// TIA Portal V16 program export: 1 tag tables, 0 data types, 1 data blocks, 11 code blocks (in call order from the OBs), 6 instance data blocks

VAR_GLOBAL   // PLC tag table "Standard-Variablentabelle"
   "Belt Conveyor (4m) 0 Encoder Signal A" AT %I0.0 : Bool;
   "Retroreflective Sensor 0" AT %I0.1 : Bool;
   "Retroreflective Sensor 1" AT %I0.2 : Bool;
   "Diffuse Sensor 0" AT %I0.3 : Bool;
   Clock_Byte AT %MB0 : Byte;
   Clock_10Hz AT %M0.0 : Bool;
   Clock_5Hz AT %M0.1 : Bool;
   "Clock_2.5Hz" AT %M0.2 : Bool;
   Clock_2Hz AT %M0.3 : Bool;
   "Clock_1.25Hz" AT %M0.4 : Bool;
   Clock_1Hz AT %M0.5 : Bool;
   "Clock_0.625Hz" AT %M0.6 : Bool;
   "Clock_0.5Hz" AT %M0.7 : Bool;
   "Diffuse Sensor 1" AT %I0.4 : Bool;
   "Diffuse Sensor 2" AT %I0.5 : Bool;
   "Diffuse Sensor 3" AT %I0.6 : Bool;
   "Belt Conveyor (2m) 0" AT %Q0.0 : Bool;
   "Belt Conveyor (2m) 1" AT %Q0.1 : Bool;
   "Belt Conveyor (2m) 2" AT %Q0.2 : Bool;
   "Belt Conveyor (2m) 3" AT %Q0.3 : Bool;
   "Belt Conveyor (4m) 0" AT %Q0.4 : Bool;
   "Conveyor Scale 0 (+)" AT %Q0.5 : Bool;
   "Pop Up Wheel Sorter 0 (+)" AT %Q0.6 : Bool;
   "Pop Up Wheel Sorter 0 (Left)" AT %Q0.7 : Bool;
   "Pop Up Wheel Sorter 0 (Right)" AT %Q1.0 : Bool;
   "Vision Sensor 0" AT %ID30 : DInt;
   Factory_Running AT %I0.7 : Bool;
   "Emergency Stop 0" AT %I1.0 : Bool;
   "Selector 0 (State 0)" AT %I1.1 : Bool;
   "Start Button 0" AT %I1.2 : Bool;
   "Two-Axis Pick & Place 0 (Detected)" AT %I1.3 : Bool;
   "Two-Axis Pick & Place 0 (Moving X)" AT %I1.4 : Bool;
   "Two-Axis Pick & Place 0 (Moving Z)" AT %I1.5 : Bool;
   "Two-Axis Pick & Place 0 X" AT %Q1.1 : Bool;
   "Two-Axis Pick & Place 0 Z" AT %Q1.2 : Bool;
   "Two-Axis Pick & Place 0 (Grab)" AT %Q1.3 : Bool;
   "Conveyor Scale 0 Weight (V)" AT %ID42 : Real;
   "Diffuse Sensor 4" AT %I1.6 : Bool;
   "Diffuse Sensor 6" AT %I1.7 : Bool;
   "Diffuse Sensor 5" AT %I2.0 : Bool;
   System_Byte AT %MB1 : Byte;
   FirstScan AT %M1.0 : Bool;
   DiagStatusUpdate AT %M1.1 : Bool;
   AlwaysTRUE AT %M1.2 : Bool;
   AlwaysFALSE AT %M1.3 : Bool;
END_VAR

DATA_BLOCK "DB_IO"   // DB1
{ S7_Optimized_Access := 'TRUE' }
VERSION : 0.1
// stored: AutoNumber true, IsOnlyStoredInLoadMemory false, IsRetainMemResEnabled false, IsWriteProtectedInAS false, MemoryReserve 100
   VAR
      One_shot : Array[0..10] of Bool;
      Green_position : DWord;
      Box_position : DWord;
      Green_raw_detected : Bool;
      System_running : Bool;
      StepA : Array[0..10] of Bool;
      Production_line_Init : Bool;
      System_Ready : Bool;
      Weight : Int;
      RunPickAndPlace : Bool;
      StepB : Array[0..10] of Bool;
      StepC : Array[0..10] of Bool;
      "counter" : Int;
   END_VAR
BEGIN
END_DATA_BLOCK

ORGANIZATION_BLOCK "Main"   // OB1, FBD, ProgramCycle
TITLE = "Main Program Sweep (Cycle)"
{ S7_Optimized_Access := 'TRUE' }
VERSION : 0.1
// stored: AutoNumber true, IsIECCheckEnabled false, SetENOAutomatically false
   VAR_INPUT
      Initial_Call : Bool;   // Initial call of this OB
      Remanence : Bool;   // =True, if remanent data are available
   END_VAR
BEGIN

REGION Network 1
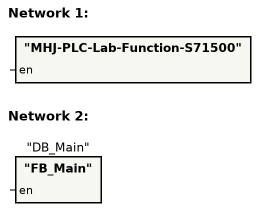
   "MHJ-PLC-Lab-Function-S71500"();
END_REGION

REGION Network 2
   "DB_Main"();   // "FB_Main"
END_REGION
END_ORGANIZATION_BLOCK

FUNCTION_BLOCK "FB_Main"   // FB2, LAD
{ S7_Optimized_Access := 'TRUE' }
VERSION : 0.1
// stored: AutoNumber true, IsIECCheckEnabled false, IsRetainMemResEnabled false, MemoryReserve 100, SetENOAutomatically false, UDAEnableTagReadback false
   VAR
      FB_Conveyor_Entry { S7_SetPoint := 'True'} : "FB_Conveyor";
      FB_Conveyor_Weight { S7_SetPoint := 'True'} : "FB_Conveyor";
      FB_WheelSorter_Instance { S7_SetPoint := 'True'} : "FB_WheelSorter";
      FB_Conveyor_Left { S7_SetPoint := 'True'} : "FB_Conveyor";
      FB_Conveyor_Straight { S7_SetPoint := 'True'} : "FB_Conveyor";
      FB_Conveyor_Right { S7_SetPoint := 'True'} : "FB_Conveyor";
      FB_PickAndPlace_Instance { S7_SetPoint := 'True'} : "FB_PickAndPlace";
      FB_Conveyor_4belt { S7_SetPoint := 'True'} : "FB_Conveyor";
   END_VAR
BEGIN

REGION Network 1
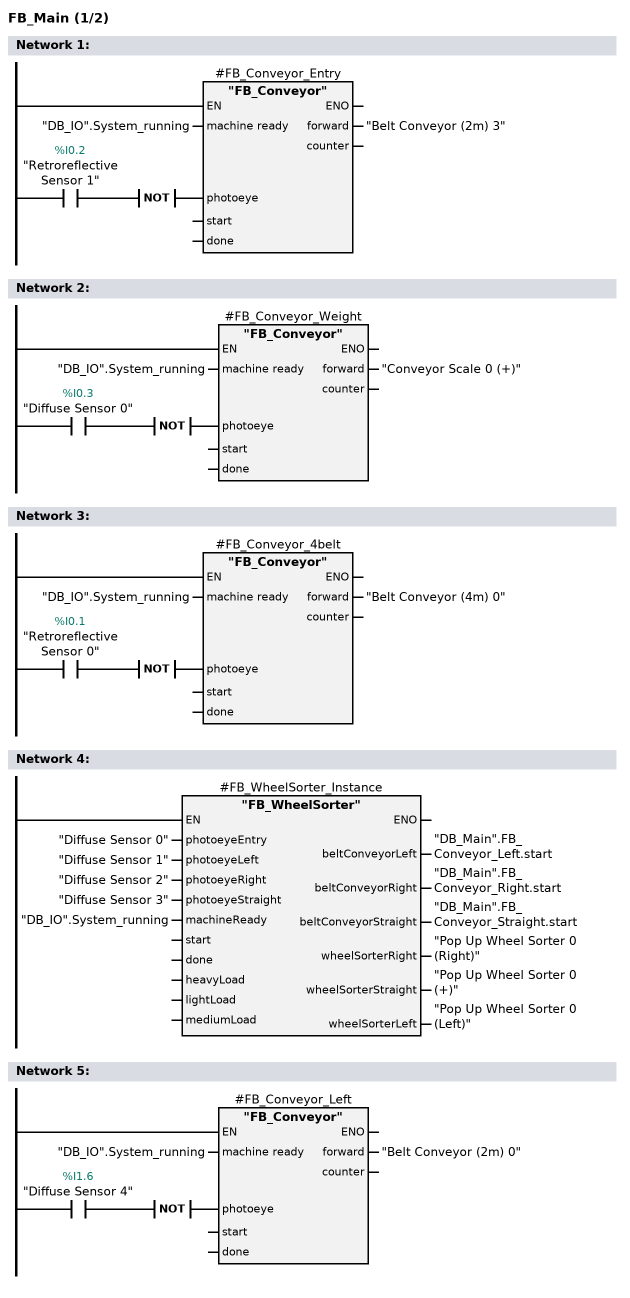
   RUNG wire#powerrail
      #FB_Conveyor_Entry(photoeye := wire#w1, "machine ready" := "DB_IO".System_running, start :=, done :=, forward => "Belt Conveyor (2m) 3", "counter" =>)
   END_RUNG
   RUNG wire#powerrail
      Contact( "Retroreflective Sensor 1" )
      Not()
   END_RUNG wire#w1
   // the same network as SCL:
   #FB_Conveyor_Entry("machine ready" := "DB_IO".System_running,   // "FB_Conveyor"
                      photoeye := NOT "Retroreflective Sensor 1",
                      forward => "Belt Conveyor (2m) 3");
END_REGION

REGION Network 2
   RUNG wire#powerrail
      #FB_Conveyor_Weight(photoeye := wire#w1, "machine ready" := "DB_IO".System_running, start :=, done :=, forward => "Conveyor Scale 0 (+)", "counter" =>)
   END_RUNG
   RUNG wire#powerrail
      Contact( "Diffuse Sensor 0" )
      Not()
   END_RUNG wire#w1
   // the same network as SCL:
   #FB_Conveyor_Weight("machine ready" := "DB_IO".System_running,   // "FB_Conveyor"
                       photoeye := NOT "Diffuse Sensor 0",
                       forward => "Conveyor Scale 0 (+)");
END_REGION

REGION Network 3
   RUNG wire#powerrail
      #FB_Conveyor_4belt(photoeye := wire#w1, "machine ready" := "DB_IO".System_running, start :=, done :=, forward => "Belt Conveyor (4m) 0", "counter" =>)
   END_RUNG
   RUNG wire#powerrail
      Contact( "Retroreflective Sensor 0" )
      Not()
   END_RUNG wire#w1
   // the same network as SCL:
   #FB_Conveyor_4belt("machine ready" := "DB_IO".System_running,   // "FB_Conveyor"
                      photoeye := NOT "Retroreflective Sensor 0",
                      forward => "Belt Conveyor (4m) 0");
END_REGION

REGION Network 4
   RUNG wire#powerrail
      #FB_WheelSorter_Instance(photoeyeEntry := "Diffuse Sensor 0", photoeyeLeft := "Diffuse Sensor 1", photoeyeRight := "Diffuse Sensor 2", photoeyeStraight := "Diffuse Sensor 3", machineReady := "DB_IO".System_running, start :=, done :=, heavyLoad :=, lightLoad :=, mediumLoad :=, beltConveyorLeft => "DB_Main".FB_Conveyor_Left.start, beltConveyorRight => "DB_Main".FB_Conveyor_Right.start, beltConveyorStraight => "DB_Main".FB_Conveyor_Straight.start, wheelSorterRight => "Pop Up Wheel Sorter 0 (Right)", wheelSorterStraight => "Pop Up Wheel Sorter 0 (+)", wheelSorterLeft => "Pop Up Wheel Sorter 0 (Left)")
   END_RUNG
   // the same network as SCL:
   #FB_WheelSorter_Instance(photoeyeEntry := "Diffuse Sensor 0",   // "FB_WheelSorter"
                           photoeyeLeft := "Diffuse Sensor 1",
                           photoeyeRight := "Diffuse Sensor 2",
                           photoeyeStraight := "Diffuse Sensor 3",
                           machineReady := "DB_IO".System_running,
                           beltConveyorLeft => "DB_Main".FB_Conveyor_Left.start,
                           beltConveyorRight => "DB_Main".FB_Conveyor_Right.start,
                           beltConveyorStraight => "DB_Main".FB_Conveyor_Straight.start,
                           wheelSorterRight => "Pop Up Wheel Sorter 0 (Right)",
                           wheelSorterStraight => "Pop Up Wheel Sorter 0 (+)",
                           wheelSorterLeft => "Pop Up Wheel Sorter 0 (Left)");
END_REGION

REGION Network 5
   RUNG wire#powerrail
      #FB_Conveyor_Left(photoeye := wire#w1, "machine ready" := "DB_IO".System_running, start :=, done :=, forward => "Belt Conveyor (2m) 0", "counter" =>)
   END_RUNG
   RUNG wire#powerrail
      Contact( "Diffuse Sensor 4" )
      Not()
   END_RUNG wire#w1
   // the same network as SCL:
   #FB_Conveyor_Left("machine ready" := "DB_IO".System_running,   // "FB_Conveyor"
                     photoeye := NOT "Diffuse Sensor 4",
                     forward => "Belt Conveyor (2m) 0");
END_REGION

REGION Network 6
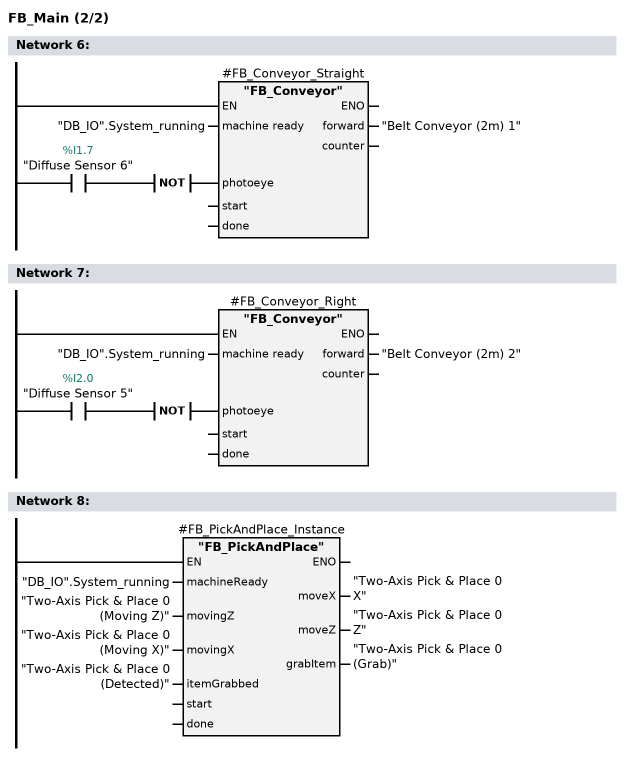
   RUNG wire#powerrail
      #FB_Conveyor_Straight(photoeye := wire#w1, "machine ready" := "DB_IO".System_running, start :=, done :=, forward => "Belt Conveyor (2m) 1", "counter" =>)
   END_RUNG
   RUNG wire#powerrail
      Contact( "Diffuse Sensor 6" )
      Not()
   END_RUNG wire#w1
   // the same network as SCL:
   #FB_Conveyor_Straight("machine ready" := "DB_IO".System_running,   // "FB_Conveyor"
                         photoeye := NOT "Diffuse Sensor 6",
                         forward => "Belt Conveyor (2m) 1");
END_REGION

REGION Network 7
   RUNG wire#powerrail
      #FB_Conveyor_Right(photoeye := wire#w1, "machine ready" := "DB_IO".System_running, start :=, done :=, forward => "Belt Conveyor (2m) 2", "counter" =>)
   END_RUNG
   RUNG wire#powerrail
      Contact( "Diffuse Sensor 5" )
      Not()
   END_RUNG wire#w1
   // the same network as SCL:
   #FB_Conveyor_Right("machine ready" := "DB_IO".System_running,   // "FB_Conveyor"
                      photoeye := NOT "Diffuse Sensor 5",
                      forward => "Belt Conveyor (2m) 2");
END_REGION

REGION Network 8
   #FB_PickAndPlace_Instance(machineReady := "DB_IO".System_running,   // "FB_PickAndPlace"
                           movingZ := "Two-Axis Pick & Place 0 (Moving Z)",
                           movingX := "Two-Axis Pick & Place 0 (Moving X)",
                           itemGrabbed := "Two-Axis Pick & Place 0 (Detected)",
                           moveX => "Two-Axis Pick & Place 0 X",
                           moveZ => "Two-Axis Pick & Place 0 Z",
                           grabItem => "Two-Axis Pick & Place 0 (Grab)");
END_REGION
END_FUNCTION_BLOCK

FUNCTION_BLOCK "FB_WheelSorter"   // FB5, LAD
{ S7_Optimized_Access := 'TRUE' }
VERSION : 0.1
// stored: AutoNumber true, IsIECCheckEnabled false, IsRetainMemResEnabled false, MemoryReserve 100, SetENOAutomatically false, UDAEnableTagReadback false
   VAR_INPUT
      photoeyeEntry : Bool;
      photoeyeLeft : Bool;
      photoeyeRight : Bool;
      photoeyeStraight : Bool;
      machineReady : Bool;
   END_VAR
   VAR_OUTPUT
      beltConveyorLeft : Bool;
      beltConveyorRight : Bool;
      beltConveyorStraight : Bool;
      wheelSorterRight : Bool;
      wheelSorterStraight : Bool;
      wheelSorterLeft : Bool;
   END_VAR
   VAR_IN_OUT
      start : Bool;
      done : Bool;
      heavyLoad : Bool := false;
      lightLoad : Bool := false;
      mediumLoad : Bool := false;
   END_VAR
   VAR
      "step" : Array[0..20] of Bool;
   END_VAR
   VAR_TEMP   // added for the SCL form of the ladder/FBD networks
      _w1 : Bool;
      _w2 : Bool;
      _w3 : Bool;
   END_VAR
BEGIN

REGION Network 1
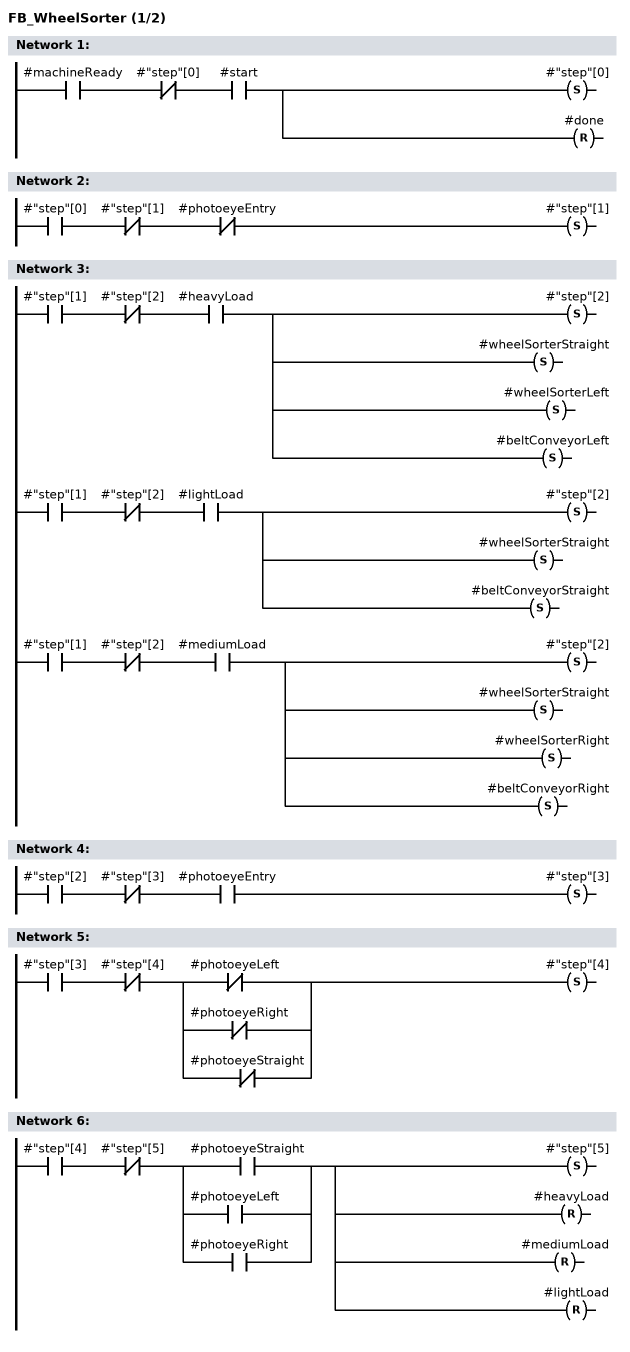
   RUNG wire#powerrail
      Contact( #machineReady )
      I_Contact( #"step"[0] )
      Contact( #start )
      wire#w1
      S_Coil( #"step"[0] )
   END_RUNG
   RUNG wire#w1
      R_Coil( #done )
   END_RUNG
   // the same network as SCL:
   #_w1 := #machineReady AND NOT #"step"[0] AND #start;
   IF #_w1 THEN
       #"step"[0] := TRUE;
       #done := FALSE;
   END_IF;
END_REGION

REGION Network 2
   RUNG wire#powerrail
      Contact( #"step"[0] )
      I_Contact( #"step"[1] )
      I_Contact( #photoeyeEntry )
      S_Coil( #"step"[1] )
   END_RUNG
   // the same network as SCL:
   IF #"step"[0] AND NOT #"step"[1] AND NOT #photoeyeEntry THEN #"step"[1] := TRUE; END_IF;
END_REGION

REGION Network 3
   RUNG wire#powerrail
      Contact( #"step"[1] )
      I_Contact( #"step"[2] )
      Contact( #heavyLoad )
      wire#w1
      S_Coil( #"step"[2] )
   END_RUNG
   RUNG wire#w1
      S_Coil( #wheelSorterStraight )
   END_RUNG
   RUNG wire#w1
      S_Coil( #wheelSorterLeft )
   END_RUNG
   RUNG wire#w1
      S_Coil( #beltConveyorLeft )
   END_RUNG
   RUNG wire#powerrail
      Contact( #"step"[1] )
      I_Contact( #"step"[2] )
      Contact( #lightLoad )
      wire#w2
      S_Coil( #"step"[2] )
   END_RUNG
   RUNG wire#w2
      S_Coil( #wheelSorterStraight )
   END_RUNG
   RUNG wire#w2
      S_Coil( #beltConveyorStraight )
   END_RUNG
   RUNG wire#powerrail
      Contact( #"step"[1] )
      I_Contact( #"step"[2] )
      Contact( #mediumLoad )
      wire#w3
      S_Coil( #"step"[2] )
   END_RUNG
   RUNG wire#w3
      S_Coil( #wheelSorterStraight )
   END_RUNG
   RUNG wire#w3
      S_Coil( #wheelSorterRight )
   END_RUNG
   RUNG wire#w3
      S_Coil( #beltConveyorRight )
   END_RUNG
   // the same network as SCL:
   #_w1 := #"step"[1] AND NOT #"step"[2] AND #heavyLoad;
   IF #_w1 THEN
       #"step"[2] := TRUE;
       #wheelSorterStraight := TRUE;
       #wheelSorterLeft := TRUE;
       #beltConveyorLeft := TRUE;
   END_IF;
   #_w2 := #"step"[1] AND NOT #"step"[2] AND #lightLoad;
   IF #_w2 THEN
       #"step"[2] := TRUE;
       #wheelSorterStraight := TRUE;
       #beltConveyorStraight := TRUE;
   END_IF;
   #_w3 := #"step"[1] AND NOT #"step"[2] AND #mediumLoad;
   IF #_w3 THEN
       #"step"[2] := TRUE;
       #wheelSorterStraight := TRUE;
       #wheelSorterRight := TRUE;
       #beltConveyorRight := TRUE;
   END_IF;
END_REGION

REGION Network 4
   RUNG wire#powerrail
      Contact( #"step"[2] )
      I_Contact( #"step"[3] )
      Contact( #photoeyeEntry )
      S_Coil( #"step"[3] )
   END_RUNG
   // the same network as SCL:
   IF #"step"[2] AND NOT #"step"[3] AND #photoeyeEntry THEN #"step"[3] := TRUE; END_IF;
END_REGION

REGION Network 5
   RUNG wire#powerrail
      Contact( #"step"[3] )
      I_Contact( #"step"[4] )
      wire#w1
      I_Contact( #photoeyeLeft )
      wire#w2
      S_Coil( #"step"[4] )
   END_RUNG
   RUNG wire#w1
      I_Contact( #photoeyeRight )
   END_RUNG wire#w2
   RUNG wire#w1
      I_Contact( #photoeyeStraight )
   END_RUNG wire#w2
   // the same network as SCL:
   IF #"step"[3] AND NOT #"step"[4] AND (NOT #photoeyeLeft OR NOT #photoeyeRight OR NOT #photoeyeStraight) THEN
       #"step"[4] := TRUE;
   END_IF;
END_REGION

REGION Network 6
   RUNG wire#powerrail
      Contact( #"step"[4] )
      I_Contact( #"step"[5] )
      wire#w1
      Contact( #photoeyeStraight )
      wire#w2
      S_Coil( #"step"[5] )
   END_RUNG
   RUNG wire#w1
      Contact( #photoeyeLeft )
   END_RUNG wire#w2
   RUNG wire#w1
      Contact( #photoeyeRight )
   END_RUNG wire#w2
   RUNG wire#w2
      R_Coil( #heavyLoad )
   END_RUNG
   RUNG wire#w2
      R_Coil( #mediumLoad )
   END_RUNG
   RUNG wire#w2
      R_Coil( #lightLoad )
   END_RUNG
   // the same network as SCL:
   #_w1 := #"step"[4] AND NOT #"step"[5] AND (#photoeyeStraight OR #photoeyeLeft OR #photoeyeRight);
   IF #_w1 THEN
       #"step"[5] := TRUE;
       #heavyLoad := FALSE;
       #mediumLoad := FALSE;
       #lightLoad := FALSE;
   END_IF;
END_REGION

REGION Network 7
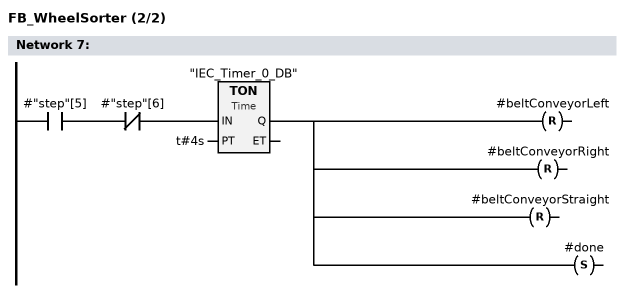
   RUNG wire#powerrail
      Contact( #"step"[5] )
      I_Contact( #"step"[6] )
      { S7_Templates := "time_type := Time" } "IEC_Timer_0_DB".TON(pt := t#4s, et =>)
      wire#w1
      R_Coil( #beltConveyorLeft )
   END_RUNG
   RUNG wire#w1
      R_Coil( #beltConveyorRight )
   END_RUNG
   RUNG wire#w1
      R_Coil( #beltConveyorStraight )
   END_RUNG
   RUNG wire#w1
      S_Coil( #done )
   END_RUNG
   // the same network as SCL:
   "IEC_Timer_0_DB".TON(IN := #"step"[5] AND NOT #"step"[6], PT := t#4s);
   IF "IEC_Timer_0_DB".Q THEN
       #beltConveyorLeft := FALSE;
       #beltConveyorRight := FALSE;
       #beltConveyorStraight := FALSE;
       #done := TRUE;
   END_IF;
END_REGION
END_FUNCTION_BLOCK

FUNCTION_BLOCK "FB_PickAndPlace"   // FB4, LAD
{ S7_Optimized_Access := 'TRUE' }
VERSION : 0.1
// stored: AutoNumber true, IsIECCheckEnabled false, IsRetainMemResEnabled false, MemoryReserve 100, SetENOAutomatically false, UDAEnableTagReadback false
   VAR_INPUT
      machineReady : Bool;
      movingZ : Bool;
      movingX : Bool;
      itemGrabbed : Bool;
   END_VAR
   VAR_OUTPUT
      moveX : Bool;
      moveZ : Bool;
      grabItem : Bool;
   END_VAR
   VAR_IN_OUT
      start : Bool;
      done : Bool;
   END_VAR
   VAR
      "step" : Array[0..20] of Bool;
   END_VAR
   VAR_TEMP   // added for the SCL form of the ladder/FBD networks
      _w1 : Bool;
   END_VAR
BEGIN

REGION Network 1: step0
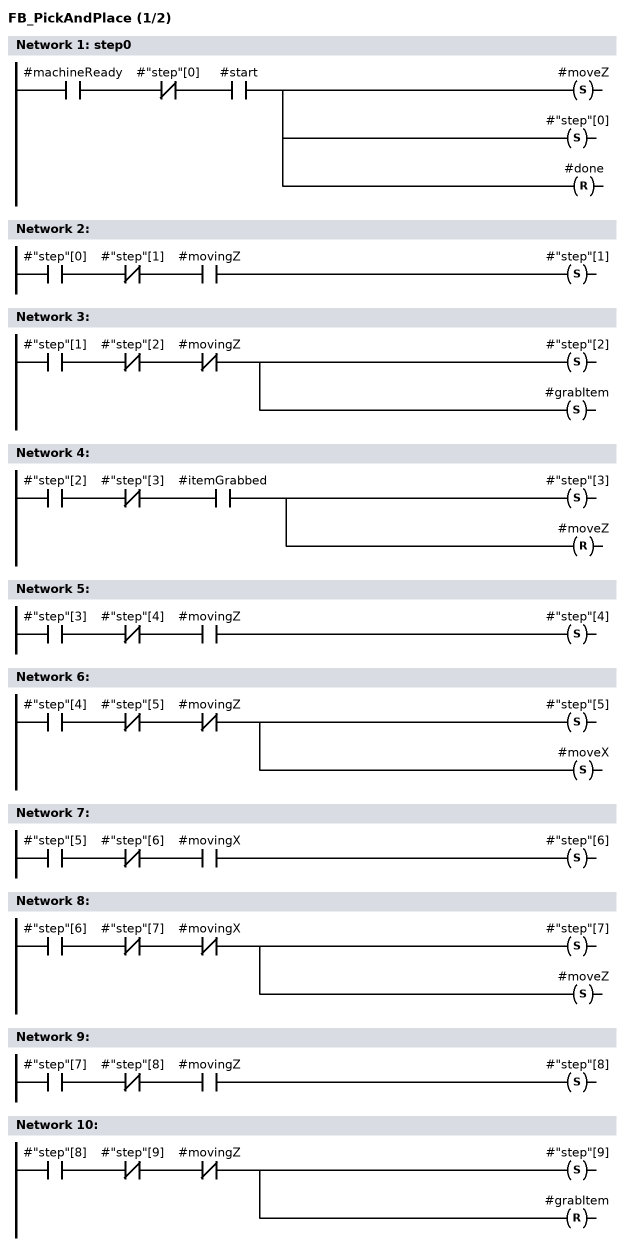
   RUNG wire#powerrail
      Contact( #machineReady )
      I_Contact( #"step"[0] )
      Contact( #start )
      wire#w1
      S_Coil( #moveZ )
   END_RUNG
   RUNG wire#w1
      S_Coil( #"step"[0] )
   END_RUNG
   RUNG wire#w1
      R_Coil( #done )
   END_RUNG
   // the same network as SCL:
   IF #machineReady AND NOT #"step"[0] AND #start THEN #moveZ := TRUE; END_IF;
   #_w1 := #machineReady AND NOT #"step"[0] AND #start;
   IF #_w1 THEN
       #"step"[0] := TRUE;
       #done := FALSE;
   END_IF;
END_REGION

REGION Network 2
   RUNG wire#powerrail
      Contact( #"step"[0] )
      I_Contact( #"step"[1] )
      Contact( #movingZ )
      S_Coil( #"step"[1] )
   END_RUNG
   // the same network as SCL:
   IF #"step"[0] AND NOT #"step"[1] AND #movingZ THEN #"step"[1] := TRUE; END_IF;
END_REGION

REGION Network 3
   RUNG wire#powerrail
      Contact( #"step"[1] )
      I_Contact( #"step"[2] )
      I_Contact( #movingZ )
      wire#w1
      S_Coil( #"step"[2] )
   END_RUNG
   RUNG wire#w1
      S_Coil( #grabItem )
   END_RUNG
   // the same network as SCL:
   #_w1 := #"step"[1] AND NOT #"step"[2] AND NOT #movingZ;
   IF #_w1 THEN
       #"step"[2] := TRUE;
       #grabItem := TRUE;
   END_IF;
END_REGION

REGION Network 4
   RUNG wire#powerrail
      Contact( #"step"[2] )
      I_Contact( #"step"[3] )
      Contact( #itemGrabbed )
      wire#w1
      S_Coil( #"step"[3] )
   END_RUNG
   RUNG wire#w1
      R_Coil( #moveZ )
   END_RUNG
   // the same network as SCL:
   #_w1 := #"step"[2] AND NOT #"step"[3] AND #itemGrabbed;
   IF #_w1 THEN
       #"step"[3] := TRUE;
       #moveZ := FALSE;
   END_IF;
END_REGION

REGION Network 5
   RUNG wire#powerrail
      Contact( #"step"[3] )
      I_Contact( #"step"[4] )
      Contact( #movingZ )
      S_Coil( #"step"[4] )
   END_RUNG
   // the same network as SCL:
   IF #"step"[3] AND NOT #"step"[4] AND #movingZ THEN #"step"[4] := TRUE; END_IF;
END_REGION

REGION Network 6
   RUNG wire#powerrail
      Contact( #"step"[4] )
      I_Contact( #"step"[5] )
      I_Contact( #movingZ )
      wire#w1
      S_Coil( #"step"[5] )
   END_RUNG
   RUNG wire#w1
      S_Coil( #moveX )
   END_RUNG
   // the same network as SCL:
   #_w1 := #"step"[4] AND NOT #"step"[5] AND NOT #movingZ;
   IF #_w1 THEN
       #"step"[5] := TRUE;
       #moveX := TRUE;
   END_IF;
END_REGION

REGION Network 7
   RUNG wire#powerrail
      Contact( #"step"[5] )
      I_Contact( #"step"[6] )
      Contact( #movingX )
      S_Coil( #"step"[6] )
   END_RUNG
   // the same network as SCL:
   IF #"step"[5] AND NOT #"step"[6] AND #movingX THEN #"step"[6] := TRUE; END_IF;
END_REGION

REGION Network 8
   RUNG wire#powerrail
      Contact( #"step"[6] )
      I_Contact( #"step"[7] )
      I_Contact( #movingX )
      wire#w1
      S_Coil( #"step"[7] )
   END_RUNG
   RUNG wire#w1
      S_Coil( #moveZ )
   END_RUNG
   // the same network as SCL:
   #_w1 := #"step"[6] AND NOT #"step"[7] AND NOT #movingX;
   IF #_w1 THEN
       #"step"[7] := TRUE;
       #moveZ := TRUE;
   END_IF;
END_REGION

REGION Network 9
   RUNG wire#powerrail
      Contact( #"step"[7] )
      I_Contact( #"step"[8] )
      Contact( #movingZ )
      S_Coil( #"step"[8] )
   END_RUNG
   // the same network as SCL:
   IF #"step"[7] AND NOT #"step"[8] AND #movingZ THEN #"step"[8] := TRUE; END_IF;
END_REGION

REGION Network 10
   RUNG wire#powerrail
      Contact( #"step"[8] )
      I_Contact( #"step"[9] )
      I_Contact( #movingZ )
      wire#w1
      S_Coil( #"step"[9] )
   END_RUNG
   RUNG wire#w1
      R_Coil( #grabItem )
   END_RUNG
   // the same network as SCL:
   #_w1 := #"step"[8] AND NOT #"step"[9] AND NOT #movingZ;
   IF #_w1 THEN
       #"step"[9] := TRUE;
       #grabItem := FALSE;
   END_IF;
END_REGION

REGION Network 11
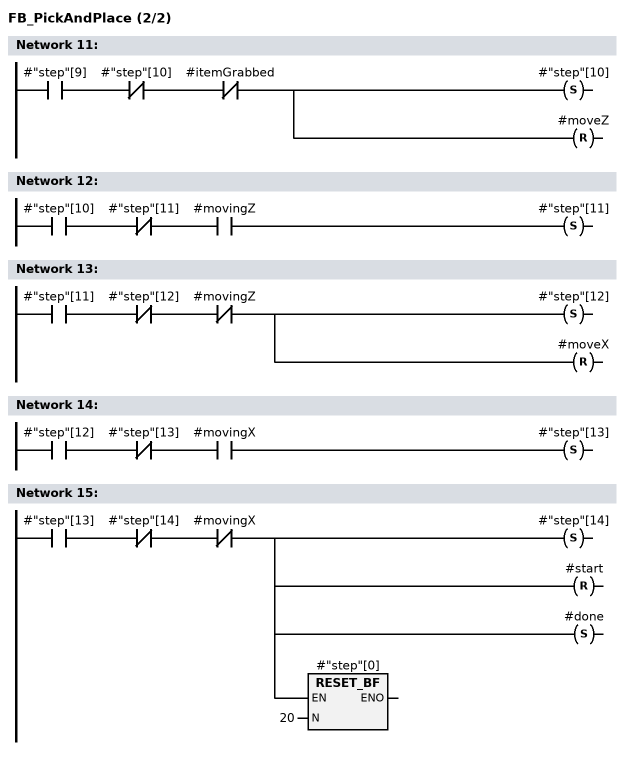
   RUNG wire#powerrail
      Contact( #"step"[9] )
      I_Contact( #"step"[10] )
      I_Contact( #itemGrabbed )
      wire#w1
      S_Coil( #"step"[10] )
   END_RUNG
   RUNG wire#w1
      R_Coil( #moveZ )
   END_RUNG
   // the same network as SCL:
   #_w1 := #"step"[9] AND NOT #"step"[10] AND NOT #itemGrabbed;
   IF #_w1 THEN
       #"step"[10] := TRUE;
       #moveZ := FALSE;
   END_IF;
END_REGION

REGION Network 12
   RUNG wire#powerrail
      Contact( #"step"[10] )
      I_Contact( #"step"[11] )
      Contact( #movingZ )
      S_Coil( #"step"[11] )
   END_RUNG
   // the same network as SCL:
   IF #"step"[10] AND NOT #"step"[11] AND #movingZ THEN #"step"[11] := TRUE; END_IF;
END_REGION

REGION Network 13
   RUNG wire#powerrail
      Contact( #"step"[11] )
      I_Contact( #"step"[12] )
      I_Contact( #movingZ )
      wire#w1
      S_Coil( #"step"[12] )
   END_RUNG
   RUNG wire#w1
      R_Coil( #moveX )
   END_RUNG
   // the same network as SCL:
   #_w1 := #"step"[11] AND NOT #"step"[12] AND NOT #movingZ;
   IF #_w1 THEN
       #"step"[12] := TRUE;
       #moveX := FALSE;
   END_IF;
END_REGION

REGION Network 14
   RUNG wire#powerrail
      Contact( #"step"[12] )
      I_Contact( #"step"[13] )
      Contact( #movingX )
      S_Coil( #"step"[13] )
   END_RUNG
   // the same network as SCL:
   IF #"step"[12] AND NOT #"step"[13] AND #movingX THEN #"step"[13] := TRUE; END_IF;
END_REGION

REGION Network 15
   // no SCL statement known for RBitfield: written as a call
   #_w1 := #"step"[13] AND NOT #"step"[14] AND NOT #movingX;
   IF #_w1 THEN
       #"step"[14] := TRUE;
       #start := FALSE;
       #done := TRUE;
       RESET_BF(operand := #"step"[0], n := 20);
   END_IF;
END_REGION
END_FUNCTION_BLOCK

ORGANIZATION_BLOCK "OB_Encoder"   // OB123, LAD, ProgramCycle
TITLE = "Main Program Sweep (Cycle)"
{ S7_Optimized_Access := 'TRUE' }
VERSION : 0.1
// stored: AutoNumber true, IsIECCheckEnabled false, SetENOAutomatically false
   VAR_INPUT
      Initial_Call : Bool;   // Initial call of this OB
      Remanence : Bool;   // =True, if remanent data are available
   END_VAR
   VAR_TEMP   // added for the SCL form of the ladder/FBD networks
      _w1 : Bool;
      _w2 : Bool;
   END_VAR
BEGIN

REGION Network 1
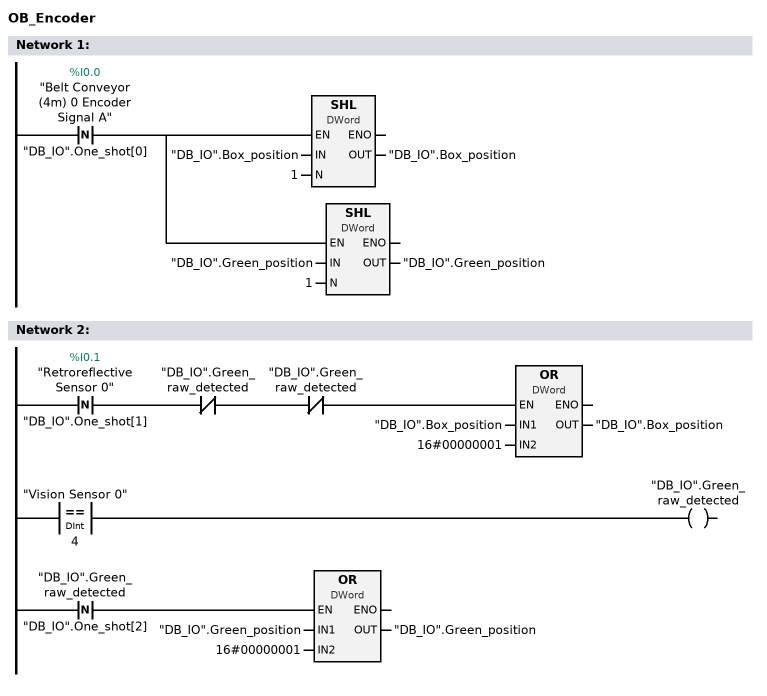
   RUNG wire#powerrail
      N_Contact(operand := "Belt Conveyor (4m) 0 Encoder Signal A", bit := "DB_IO".One_shot[0])
      wire#w1
      { S7_Templates := "SrcType := DWord" } Shl(in := "DB_IO".Box_position, n := 1, out => "DB_IO".Box_position)
   END_RUNG
   RUNG wire#w1
      { S7_Templates := "SrcType := DWord" } Shl(in := "DB_IO".Green_position, n := 1, out => "DB_IO".Green_position)
   END_RUNG
   // the same network as SCL:
   #_w1 := NOT "Belt Conveyor (4m) 0 Encoder Signal A" AND "DB_IO".One_shot[0];   // falling edge of "Belt Conveyor (4m) 0 Encoder Signal A"
   "DB_IO".One_shot[0] := "Belt Conveyor (4m) 0 Encoder Signal A";
   IF #_w1 THEN
       "DB_IO".Box_position := SHL(IN := "DB_IO".Box_position, N := 1);
       "DB_IO".Green_position := SHL(IN := "DB_IO".Green_position, N := 1);
   END_IF;
END_REGION

REGION Network 2
   #_w1 := NOT "Retroreflective Sensor 0" AND "DB_IO".One_shot[1];   // falling edge of "Retroreflective Sensor 0"
   "DB_IO".One_shot[1] := "Retroreflective Sensor 0";
   IF #_w1 AND NOT "DB_IO".Green_raw_detected AND NOT "DB_IO".Green_raw_detected THEN
       "DB_IO".Box_position := "DB_IO".Box_position OR 16#00000001;
   END_IF;
   "DB_IO".Green_raw_detected := "Vision Sensor 0" = 4;
   #_w2 := NOT "DB_IO".Green_raw_detected AND "DB_IO".One_shot[2];   // falling edge of "DB_IO".Green_raw_detected
   "DB_IO".One_shot[2] := "DB_IO".Green_raw_detected;
   IF #_w2 THEN "DB_IO".Green_position := "DB_IO".Green_position OR 16#00000001; END_IF;
END_REGION
END_ORGANIZATION_BLOCK

ORGANIZATION_BLOCK "OB_Line_Init"   // OB125, LAD, ProgramCycle
TITLE = "Main Program Sweep (Cycle)"
{ S7_Optimized_Access := 'TRUE' }
VERSION : 0.1
// stored: AutoNumber true, IsIECCheckEnabled false, SetENOAutomatically false
   VAR_INPUT
      Initial_Call : Bool;   // Initial call of this OB
      Remanence : Bool;   // =True, if remanent data are available
   END_VAR
   VAR_TEMP   // added for the SCL form of the ladder/FBD networks
      _w1 : Bool;
   END_VAR
BEGIN

REGION Network 1
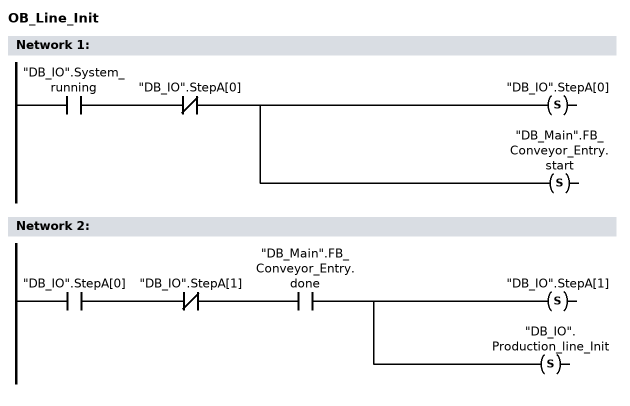
   RUNG wire#powerrail
      Contact( "DB_IO".System_running )
      I_Contact( "DB_IO".StepA[0] )
      wire#w1
      S_Coil( "DB_IO".StepA[0] )
   END_RUNG
   RUNG wire#w1
      S_Coil( "DB_Main".FB_Conveyor_Entry.start )
   END_RUNG
   // the same network as SCL:
   #_w1 := "DB_IO".System_running AND NOT "DB_IO".StepA[0];
   IF #_w1 THEN
       "DB_IO".StepA[0] := TRUE;
       "DB_Main".FB_Conveyor_Entry.start := TRUE;
   END_IF;
END_REGION

REGION Network 2
   RUNG wire#powerrail
      Contact( "DB_IO".StepA[0] )
      I_Contact( "DB_IO".StepA[1] )
      Contact( "DB_Main".FB_Conveyor_Entry.done )
      wire#w1
      S_Coil( "DB_IO".StepA[1] )
   END_RUNG
   RUNG wire#w1
      S_Coil( "DB_IO".Production_line_Init )
   END_RUNG
   // the same network as SCL:
   #_w1 := "DB_IO".StepA[0] AND NOT "DB_IO".StepA[1] AND "DB_Main".FB_Conveyor_Entry.done;
   IF #_w1 THEN
       "DB_IO".StepA[1] := TRUE;
       "DB_IO".Production_line_Init := TRUE;
   END_IF;
END_REGION
END_ORGANIZATION_BLOCK

ORGANIZATION_BLOCK "OB_Machine_Ready"   // OB126, LAD, ProgramCycle
TITLE = "Main Program Sweep (Cycle)"
{ S7_Optimized_Access := 'TRUE' }
VERSION : 0.1
// stored: AutoNumber true, IsIECCheckEnabled false, SetENOAutomatically false
   VAR_INPUT
      Initial_Call : Bool;   // Initial call of this OB
      Remanence : Bool;   // =True, if remanent data are available
   END_VAR
BEGIN

REGION Network 1
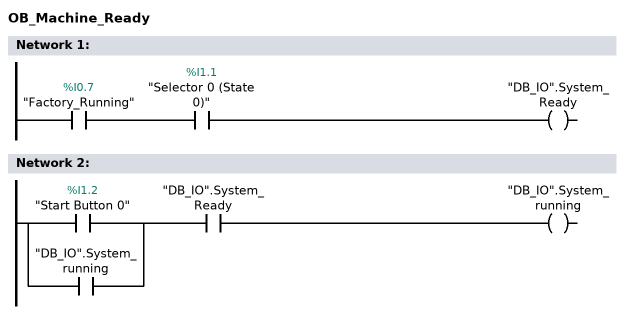
   RUNG wire#powerrail
      Contact( "Factory_Running" )
      Contact( "Selector 0 (State 0)" )
      Coil( "DB_IO".System_Ready )
   END_RUNG
   // the same network as SCL:
   "DB_IO".System_Ready := "Factory_Running" AND "Selector 0 (State 0)";
END_REGION

REGION Network 2
   RUNG wire#powerrail
      Contact( "Start Button 0" )
      wire#w1
      Contact( "DB_IO".System_Ready )
      Coil( "DB_IO".System_running )
   END_RUNG
   RUNG wire#powerrail
      Contact( "DB_IO".System_running )
   END_RUNG wire#w1
   // the same network as SCL:
   "DB_IO".System_running := ("Start Button 0" OR "DB_IO".System_running) AND "DB_IO".System_Ready;
END_REGION
END_ORGANIZATION_BLOCK

ORGANIZATION_BLOCK "OB_Master"   // OB124, LAD, ProgramCycle
TITLE = "Main Program Sweep (Cycle)"
{ S7_Optimized_Access := 'TRUE' }
VERSION : 0.1
// stored: AutoNumber true, IsIECCheckEnabled false, SetENOAutomatically false
   VAR_INPUT
      Initial_Call : Bool;   // Initial call of this OB
      Remanence : Bool;   // =True, if remanent data are available
   END_VAR
BEGIN

REGION Network 1
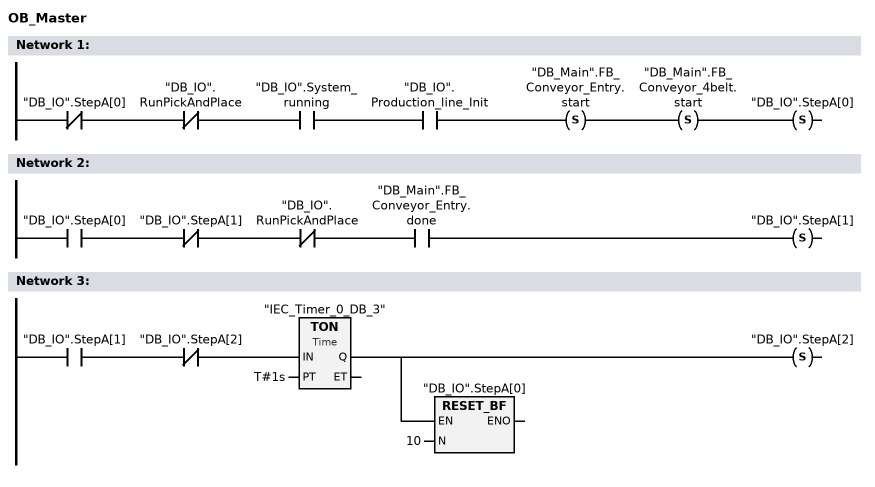
   RUNG wire#powerrail
      I_Contact( "DB_IO".StepA[0] )
      I_Contact( "DB_IO".RunPickAndPlace )
      Contact( "DB_IO".System_running )
      Contact( "DB_IO".Production_line_Init )
      S_Coil( "DB_Main".FB_Conveyor_Entry.start )
      S_Coil( "DB_Main".FB_Conveyor_4belt.start )
      S_Coil( "DB_IO".StepA[0] )
   END_RUNG
   // the same network as SCL:
   IF NOT "DB_IO".StepA[0] AND NOT "DB_IO".RunPickAndPlace AND "DB_IO".System_running AND "DB_IO".Production_line_Init THEN
       "DB_Main".FB_Conveyor_Entry.start := TRUE;
       "DB_Main".FB_Conveyor_4belt.start := TRUE;
       "DB_IO".StepA[0] := TRUE;
   END_IF;
END_REGION

REGION Network 2
   RUNG wire#powerrail
      Contact( "DB_IO".StepA[0] )
      I_Contact( "DB_IO".StepA[1] )
      I_Contact( "DB_IO".RunPickAndPlace )
      Contact( "DB_Main".FB_Conveyor_Entry.done )
      S_Coil( "DB_IO".StepA[1] )
   END_RUNG
   // the same network as SCL:
   IF "DB_IO".StepA[0] AND NOT "DB_IO".StepA[1] AND NOT "DB_IO".RunPickAndPlace AND "DB_Main".FB_Conveyor_Entry.done THEN
       "DB_IO".StepA[1] := TRUE;
   END_IF;
END_REGION

REGION Network 3
   // no SCL statement known for RBitfield: written as a call
   "IEC_Timer_0_DB_3".TON(IN := "DB_IO".StepA[1] AND NOT "DB_IO".StepA[2], PT := T#1s);
   IF "IEC_Timer_0_DB_3".Q THEN
       "DB_IO".StepA[2] := TRUE;
       RESET_BF(operand := "DB_IO".StepA[0], n := 10);
   END_IF;
END_REGION
END_ORGANIZATION_BLOCK

ORGANIZATION_BLOCK "OB_PickAndPlace"   // OB127, LAD, ProgramCycle
TITLE = "Main Program Sweep (Cycle)"
{ S7_Optimized_Access := 'TRUE' }
VERSION : 0.1
// stored: AutoNumber true, IsIECCheckEnabled false, SetENOAutomatically false
   VAR_INPUT
      Initial_Call : Bool;   // Initial call of this OB
      Remanence : Bool;   // =True, if remanent data are available
   END_VAR
   VAR_TEMP   // added for the SCL form of the ladder/FBD networks
      _w1 : Bool;
   END_VAR
BEGIN

REGION Network 1
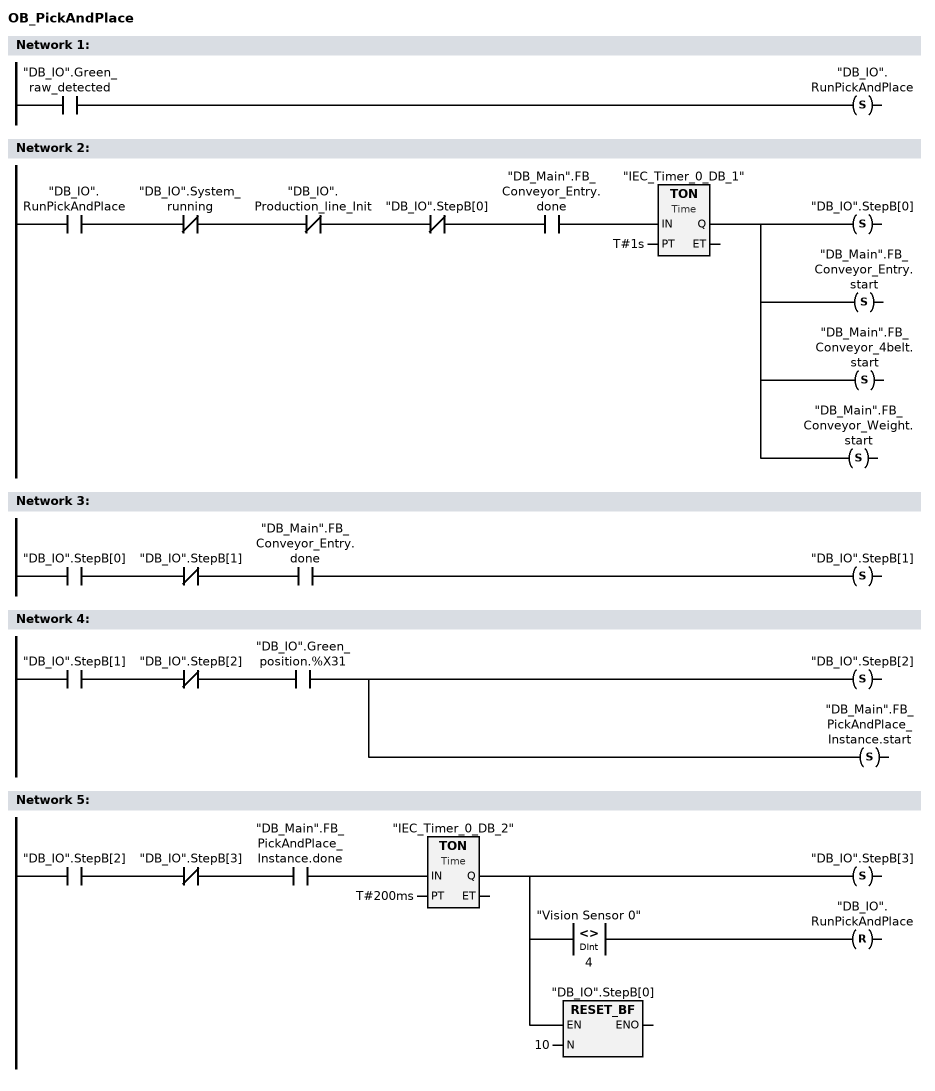
   RUNG wire#powerrail
      Contact( "DB_IO".Green_raw_detected )
      S_Coil( "DB_IO".RunPickAndPlace )
   END_RUNG
   // the same network as SCL:
   IF "DB_IO".Green_raw_detected THEN "DB_IO".RunPickAndPlace := TRUE; END_IF;
END_REGION

REGION Network 2
   RUNG wire#powerrail
      Contact( "DB_IO".RunPickAndPlace )
      I_Contact( "DB_IO".System_running )
      I_Contact( "DB_IO".Production_line_Init )
      I_Contact( "DB_IO".StepB[0] )
      Contact( "DB_Main".FB_Conveyor_Entry.done )
      { S7_Templates := "time_type := Time" } "IEC_Timer_0_DB_1".TON(pt := T#1s, et =>)
      wire#w1
      S_Coil( "DB_IO".StepB[0] )
   END_RUNG
   RUNG wire#w1
      S_Coil( "DB_Main".FB_Conveyor_Entry.start )
   END_RUNG
   RUNG wire#w1
      S_Coil( "DB_Main".FB_Conveyor_4belt.start )
   END_RUNG
   RUNG wire#w1
      S_Coil( "DB_Main".FB_Conveyor_Weight.start )
   END_RUNG
   // the same network as SCL:
   "IEC_Timer_0_DB_1".TON(IN := "DB_IO".RunPickAndPlace AND NOT "DB_IO".System_running AND NOT "DB_IO".Production_line_Init AND NOT "DB_IO".StepB[0] AND "DB_Main".FB_Conveyor_Entry.done,
                          PT := T#1s);
   IF "IEC_Timer_0_DB_1".Q THEN
       "DB_IO".StepB[0] := TRUE;
       "DB_Main".FB_Conveyor_Entry.start := TRUE;
       "DB_Main".FB_Conveyor_4belt.start := TRUE;
       "DB_Main".FB_Conveyor_Weight.start := TRUE;
   END_IF;
END_REGION

REGION Network 3
   RUNG wire#powerrail
      Contact( "DB_IO".StepB[0] )
      I_Contact( "DB_IO".StepB[1] )
      Contact( "DB_Main".FB_Conveyor_Entry.done )
      S_Coil( "DB_IO".StepB[1] )
   END_RUNG
   // the same network as SCL:
   IF "DB_IO".StepB[0] AND NOT "DB_IO".StepB[1] AND "DB_Main".FB_Conveyor_Entry.done THEN
       "DB_IO".StepB[1] := TRUE;
   END_IF;
END_REGION

REGION Network 4
   RUNG wire#powerrail
      Contact( "DB_IO".StepB[1] )
      I_Contact( "DB_IO".StepB[2] )
      Contact( "DB_IO".Green_position.%X31 )
      wire#w1
      S_Coil( "DB_IO".StepB[2] )
   END_RUNG
   RUNG wire#w1
      S_Coil( "DB_Main".FB_PickAndPlace_Instance.start )
   END_RUNG
   // the same network as SCL:
   #_w1 := "DB_IO".StepB[1] AND NOT "DB_IO".StepB[2] AND "DB_IO".Green_position.%X31;
   IF #_w1 THEN
       "DB_IO".StepB[2] := TRUE;
       "DB_Main".FB_PickAndPlace_Instance.start := TRUE;
   END_IF;
END_REGION

REGION Network 5
   // no SCL statement known for RBitfield: written as a call
   "IEC_Timer_0_DB_2".TON(IN := "DB_IO".StepB[2] AND NOT "DB_IO".StepB[3] AND "DB_Main".FB_PickAndPlace_Instance.done,
                          PT := T#200ms);
   IF "IEC_Timer_0_DB_2".Q THEN "DB_IO".StepB[3] := TRUE; END_IF;
   IF "IEC_Timer_0_DB_2".Q AND ("Vision Sensor 0" <> 4) THEN "DB_IO".RunPickAndPlace := FALSE; END_IF;
   IF "IEC_Timer_0_DB_2".Q THEN RESET_BF(operand := "DB_IO".StepB[0], n := 10); END_IF;
END_REGION
END_ORGANIZATION_BLOCK

ORGANIZATION_BLOCK "OB_WeightSorter"   // OB128, LAD, ProgramCycle
TITLE = "Main Program Sweep (Cycle)"
{ S7_Optimized_Access := 'TRUE' }
VERSION : 0.1
// stored: AutoNumber true, IsIECCheckEnabled false, SetENOAutomatically false
   VAR_INPUT
      Initial_Call : Bool;   // Initial call of this OB
      Remanence : Bool;   // =True, if remanent data are available
   END_VAR
   VAR_TEMP   // added for the SCL form of the ladder/FBD networks
      _w1 : Bool;
   END_VAR
BEGIN

REGION Network 1
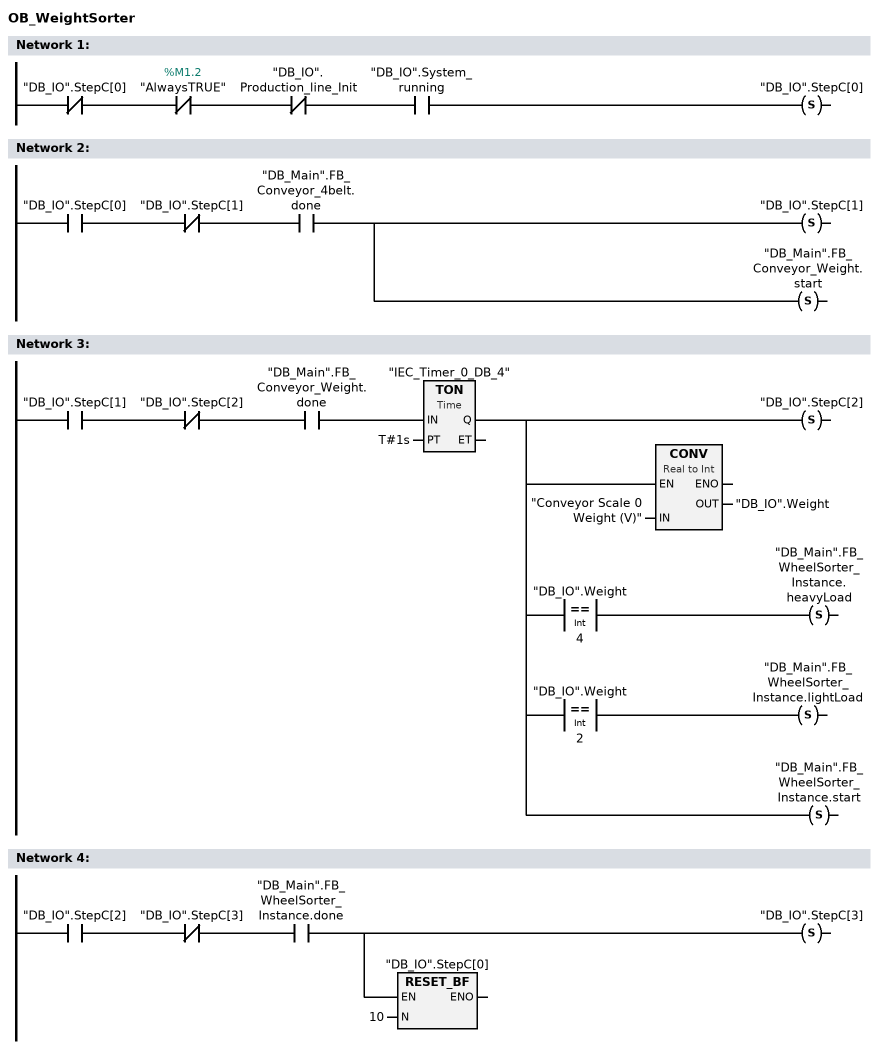
   RUNG wire#powerrail
      I_Contact( "DB_IO".StepC[0] )
      I_Contact( "AlwaysTRUE" )
      I_Contact( "DB_IO".Production_line_Init )
      Contact( "DB_IO".System_running )
      S_Coil( "DB_IO".StepC[0] )
   END_RUNG
   // the same network as SCL:
   IF NOT "DB_IO".StepC[0] AND NOT "AlwaysTRUE" AND NOT "DB_IO".Production_line_Init AND "DB_IO".System_running THEN
       "DB_IO".StepC[0] := TRUE;
   END_IF;
END_REGION

REGION Network 2
   RUNG wire#powerrail
      Contact( "DB_IO".StepC[0] )
      I_Contact( "DB_IO".StepC[1] )
      Contact( "DB_Main".FB_Conveyor_4belt.done )
      wire#w1
      S_Coil( "DB_IO".StepC[1] )
   END_RUNG
   RUNG wire#w1
      S_Coil( "DB_Main".FB_Conveyor_Weight.start )
   END_RUNG
   // the same network as SCL:
   #_w1 := "DB_IO".StepC[0] AND NOT "DB_IO".StepC[1] AND "DB_Main".FB_Conveyor_4belt.done;
   IF #_w1 THEN
       "DB_IO".StepC[1] := TRUE;
       "DB_Main".FB_Conveyor_Weight.start := TRUE;
   END_IF;
END_REGION

REGION Network 3
   RUNG wire#powerrail
      Contact( "DB_IO".StepC[1] )
      I_Contact( "DB_IO".StepC[2] )
      Contact( "DB_Main".FB_Conveyor_Weight.done )
      { S7_Templates := "time_type := Time" } "IEC_Timer_0_DB_4".TON(pt := T#1s, et =>)
      wire#w1
      S_Coil( "DB_IO".StepC[2] )
   END_RUNG
   RUNG wire#w1
      { S7_Templates := "[SrcType := Real, DestType := Int]" } Convert(in := "Conveyor Scale 0 Weight (V)", out => "DB_IO".Weight)
   END_RUNG
   RUNG wire#w1
      { S7_Templates := "SrcType := Int" } EQ_Contact(in1 := "DB_IO".Weight, in2 := 4)
      S_Coil( "DB_Main".FB_WheelSorter_Instance.heavyLoad )
   END_RUNG
   RUNG wire#w1
      { S7_Templates := "SrcType := Int" } EQ_Contact(in1 := "DB_IO".Weight, in2 := 2)
      S_Coil( "DB_Main".FB_WheelSorter_Instance.lightLoad )
   END_RUNG
   RUNG wire#w1
      S_Coil( "DB_Main".FB_WheelSorter_Instance.start )
   END_RUNG
   // the same network as SCL:
   "IEC_Timer_0_DB_4".TON(IN := "DB_IO".StepC[1] AND NOT "DB_IO".StepC[2] AND "DB_Main".FB_Conveyor_Weight.done,
                          PT := T#1s);
   IF "IEC_Timer_0_DB_4".Q THEN
       "DB_IO".StepC[2] := TRUE;
       "DB_IO".Weight := REAL_TO_INT("Conveyor Scale 0 Weight (V)");
   END_IF;
   IF "IEC_Timer_0_DB_4".Q AND ("DB_IO".Weight = 4) THEN
       "DB_Main".FB_WheelSorter_Instance.heavyLoad := TRUE;
   END_IF;
   IF "IEC_Timer_0_DB_4".Q AND ("DB_IO".Weight = 2) THEN
       "DB_Main".FB_WheelSorter_Instance.lightLoad := TRUE;
   END_IF;
   IF "IEC_Timer_0_DB_4".Q THEN "DB_Main".FB_WheelSorter_Instance.start := TRUE; END_IF;
END_REGION

REGION Network 4
   // no SCL statement known for RBitfield: written as a call
   #_w1 := "DB_IO".StepC[2] AND NOT "DB_IO".StepC[3] AND "DB_Main".FB_WheelSorter_Instance.done;
   IF #_w1 THEN
       "DB_IO".StepC[3] := TRUE;
       RESET_BF(operand := "DB_IO".StepC[0], n := 10);
   END_IF;
END_REGION
END_ORGANIZATION_BLOCK

FUNCTION_BLOCK "FB_Pusher"   // FB1, LAD
{ S7_Optimized_Access := 'TRUE' }
VERSION : 0.1
// stored: AutoNumber true, IsIECCheckEnabled false, IsRetainMemResEnabled false, MemoryReserve 100, SetENOAutomatically false, UDAEnableTagReadback false
   VAR_INPUT
      "machine ready" : Bool;
      "front limit" : Bool;
      "back limit" : Bool;
   END_VAR
   VAR_OUTPUT
      extend : Bool;
      "counter" : Bool;
   END_VAR
   VAR_IN_OUT
      start : Bool;
      done : Bool;
   END_VAR
   VAR
      "step" : Array[0..19] of Bool;
   END_VAR
   VAR_TEMP   // added for the SCL form of the ladder/FBD networks
      _w1 : Bool;
   END_VAR
BEGIN

REGION Network 1
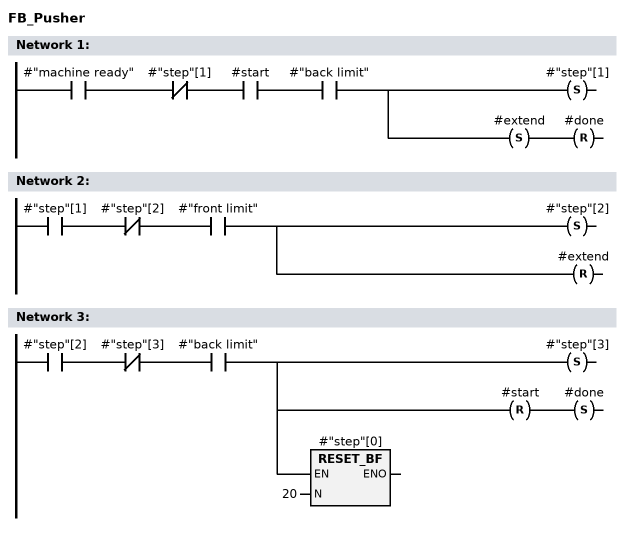
   RUNG wire#powerrail
      Contact( #"machine ready" )
      I_Contact( #"step"[1] )
      Contact( #start )
      Contact( #"back limit" )
      wire#w1
      S_Coil( #"step"[1] )
   END_RUNG
   RUNG wire#w1
      S_Coil( #extend )
      R_Coil( #done )
   END_RUNG
   // the same network as SCL:
   #_w1 := #"machine ready" AND NOT #"step"[1] AND #start AND #"back limit";
   IF #_w1 THEN
       #"step"[1] := TRUE;
       #extend := TRUE;
       #done := FALSE;
   END_IF;
END_REGION

REGION Network 2
   RUNG wire#powerrail
      Contact( #"step"[1] )
      I_Contact( #"step"[2] )
      Contact( #"front limit" )
      wire#w1
      S_Coil( #"step"[2] )
   END_RUNG
   RUNG wire#w1
      R_Coil( #extend )
   END_RUNG
   // the same network as SCL:
   #_w1 := #"step"[1] AND NOT #"step"[2] AND #"front limit";
   IF #_w1 THEN
       #"step"[2] := TRUE;
       #extend := FALSE;
   END_IF;
END_REGION

REGION Network 3
   // no SCL statement known for RBitfield: written as a call
   #_w1 := #"step"[2] AND NOT #"step"[3] AND #"back limit";
   IF #_w1 THEN
       #"step"[3] := TRUE;
       #start := FALSE;
       #done := TRUE;
       RESET_BF(operand := #"step"[0], n := 20);
   END_IF;
END_REGION
END_FUNCTION_BLOCK

DATA_BLOCK "DB_Main"   // DB2
VERSION : 0.1
// stored: AutoNumber true, InstanceOfName FB_Main, InstanceOfType FB
"FB_Main"
BEGIN
END_DATA_BLOCK

DATA_BLOCK "IEC_Timer_0_DB"   // DB4
{ S7_Optimized_Access := 'TRUE' }
// stored: AutoNumber true, InstanceOfName IEC_TIMER, OfSystemLibElement IEC_TIMER, OfSystemLibVersion 1.0
"IEC_TIMER"
   // VAR
   //    PT : Time;
   //    ET { ExternalWritable := 'False'} : Time;
   //    IN : Bool;
   //    Q { ExternalWritable := 'False'} : Bool;
   // END_VAR
BEGIN
END_DATA_BLOCK

DATA_BLOCK "IEC_Timer_0_DB_1"   // DB3
{ S7_Optimized_Access := 'TRUE' }
// stored: AutoNumber true, InstanceOfName IEC_TIMER, OfSystemLibElement IEC_TIMER, OfSystemLibVersion 1.0
"IEC_TIMER"
   // VAR
   //    PT : Time;
   //    ET { ExternalWritable := 'False'} : Time;
   //    IN : Bool;
   //    Q { ExternalWritable := 'False'} : Bool;
   // END_VAR
BEGIN
END_DATA_BLOCK

DATA_BLOCK "IEC_Timer_0_DB_2"   // DB5
{ S7_Optimized_Access := 'TRUE' }
// stored: AutoNumber true, InstanceOfName IEC_TIMER, OfSystemLibElement IEC_TIMER, OfSystemLibVersion 1.0
"IEC_TIMER"
   // VAR
   //    PT : Time;
   //    ET { ExternalWritable := 'False'} : Time;
   //    IN : Bool;
   //    Q { ExternalWritable := 'False'} : Bool;
   // END_VAR
BEGIN
END_DATA_BLOCK

DATA_BLOCK "IEC_Timer_0_DB_3"   // DB6
{ S7_Optimized_Access := 'TRUE' }
// stored: AutoNumber true, InstanceOfName IEC_TIMER, OfSystemLibElement IEC_TIMER, OfSystemLibVersion 1.0
"IEC_TIMER"
   // VAR
   //    PT : Time;
   //    ET { ExternalWritable := 'False'} : Time;
   //    IN : Bool;
   //    Q { ExternalWritable := 'False'} : Bool;
   // END_VAR
BEGIN
END_DATA_BLOCK

DATA_BLOCK "IEC_Timer_0_DB_4"   // DB7
{ S7_Optimized_Access := 'TRUE' }
// stored: AutoNumber true, InstanceOfName IEC_TIMER, OfSystemLibElement IEC_TIMER, OfSystemLibVersion 1.0
"IEC_TIMER"
   // VAR
   //    PT : Time;
   //    ET { ExternalWritable := 'False'} : Time;
   //    IN : Bool;
   //    Q { ExternalWritable := 'False'} : Bool;
   // END_VAR
BEGIN
END_DATA_BLOCK
